FUNCTION_BLOCK SafetyStopBasic (* Basic Function Block Type *)
  (* Standard: 61499-2 *)
  (* Version 0.0, 6/17/2024, SESA713705, Schneider Electric, Template *)
  PACKAGE SE.Nereda;
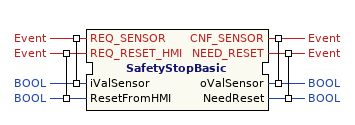
  EVENT_INPUT
    REQ_SENSOR WITH iValSensor;
    REQ_RESET_HMI WITH ResetFromHMI;
  END_EVENT
  EVENT_OUTPUT
    CNF_SENSOR WITH oValSensor;
    NEED_RESET WITH NeedReset;
  END_EVENT
  VAR_INPUT
    iValSensor : BOOL;
    ResetFromHMI : BOOL;
  END_VAR
  VAR_OUTPUT
    oValSensor : BOOL;
    NeedReset : BOOL;
  END_VAR
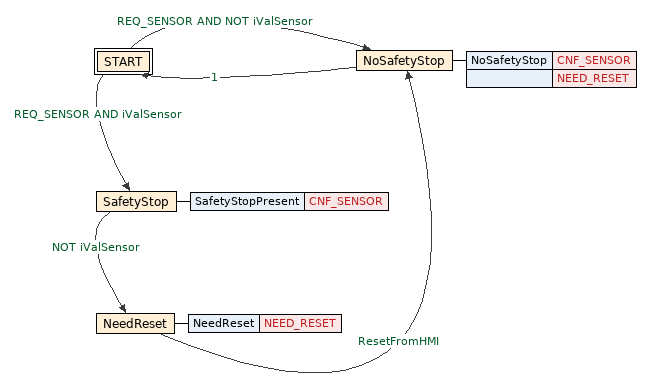
  EC_STATES
    START; (* Initial State *)
    NoSafetyStop : NoSafetyStop -> CNF_SENSOR, -> NEED_RESET;
    SafetyStop : SafetyStopPresent -> CNF_SENSOR;
    NeedReset : NeedReset -> NEED_RESET;
  END_STATES
  EC_TRANSITIONS
    START TO NoSafetyStop := REQ_SENSOR AND NOT iValSensor;
    NoSafetyStop TO START := 1;
    START TO SafetyStop := REQ_SENSOR AND iValSensor;
    SafetyStop TO NeedReset := NOT iValSensor;
    NeedReset TO NoSafetyStop := ResetFromHMI;
  END_TRANSITIONS
  ALGORITHM NoSafetyStop IN ST:
;
oValSensor := iValSensor;
NeedReset := FALSE;
  END_ALGORITHM
  ALGORITHM SafetyStopPresent IN ST:
;
oValSensor := iValSensor;
  END_ALGORITHM
  ALGORITHM NeedReset IN ST:
;
NeedReset := TRUE;
  END_ALGORITHM
END_FUNCTION_BLOCK
